// TIA Portal project "AB" (V15.1)

(* hardware
DEVICE "S71500/ET200MP station_1"  S7-1500 station
   slot 0: "导轨_0"  Rack  6ES7 590-1***0-0AA0
   slot 0: "PS 25W 24VDC_1"  PS 25W 24VDC  6ES7 505-0KA00-0AB0  V1.0
   slot 1: "PLC_1"  CPU 1515-2 PN  6ES7 515-2AM01-0AB0  V2.6
      slot 3: "CPU 显示_1"  6ES7591-1BA00-0AA0
DEVICE "HMI_1"  TP900 Comfort
   slot 0: "HMI_1"  TP900 Comfort  6AV2 124-0JC01-0AX0  15.1.0.0
   slot 1: "HMI_RT_1"  TP900 Comfort  6AV2 124-0JC01-0AX0  15.1.0.0
   slot 5: "HMI_1.IE_CP_1"  PROFINET Interface  15.0.1.0
      slot 1: "PROFINET Interface_1"  PROFINET Interface
         slot 1: "Port_1"  Port
         slot 2: "Port_2"  Port
   slot 7: "HMI_1.MPI/DP_CP_1"  MPI/DP Interface  15.0.1.0
*)

// ===== PLC "PLC_1"  CPU 1515-2 PN =====

VAR_GLOBAL   // PLC tag table "默认变量表"
   "System_Byte" AT %MB1 : Byte;
   "FirstScan" AT %M1.0 : Bool;
   "DiagStatusUpdate" AT %M1.1 : Bool;
   "AlwaysTRUE" AT %M1.2 : Bool;
   "AlwaysFALSE" AT %M1.3 : Bool;
   "Clock_Byte" AT %MB0 : Byte;
   "Clock_10Hz" AT %M0.0 : Bool;
   "Clock_5Hz" AT %M0.1 : Bool;
   "Clock_2.5Hz" AT %M0.2 : Bool;
   "Clock_2Hz" AT %M0.3 : Bool;
   "Clock_1.25Hz" AT %M0.4 : Bool;
   "Clock_1Hz" AT %M0.5 : Bool;
   "Clock_0.625Hz" AT %M0.6 : Bool;
   "Clock_0.5Hz" AT %M0.7 : Bool;
END_VAR

TYPE "Motor"
   STRUCT
      运行时间 : Time;   // 电机连续运行时间
      输出频率 : Real;   // 电机变频器当前输出频率
      A相电压 : Real;   // 变频器当前A相电压
      B相电压 : Real;   // 变频器当前B相电压
      C相电压 : Real;   // 变频器当前C相电压
      A相电流 : Real;   // 变频器当前A相电流
      B相电流 : Real;   // 变频器当前B相电流
      C相电流 : Real;   // 变频器当前C相电流
      启动 : Bool;   // 启动指令
      停止 : Bool;   // 停止指令
   END_STRUCT;
END_TYPE

DATA_BLOCK "_DeBug"   // DB1
{ S7_Optimized_Access := 'FALSE' }
VERSION : 0.1
   VAR
      IN : Word;
      max : Real;
      min : Real;
      amax : Int;
      amin : Int;
      error : Bool;
      status : Word;
      ret : Real;
      "1err" : Bool;
      "1sta" : Word;
      "1ot" : Word;
      计数 : Bool;
      temp : Array[0..1] of Bool;
      次数 : Int;
   END_VAR
BEGIN
END_DATA_BLOCK

// folder: 500 Communication

DATA_BLOCK "ConnectSet"   // DB501
{ S7_Optimized_Access := 'FALSE' }
VERSION : 0.1
   VAR
      connect : TCON_IP_v4;
   END_VAR
BEGIN
   connect.InterfaceId := 64;
   connect.ID := 1;
   connect.LocalPort := 502;
END_DATA_BLOCK

// folder: 500 Communication/PLCtoUpper

DATA_BLOCK "CommData_0x"   // DB503
{ S7_Optimized_Access := 'FALSE' }
VERSION : 0.1
   VAR
      "1-1#阀门" : Bool;   // 00001
      "1-2#阀门" : Bool;   // 00002
      "1-3#阀门" : Bool;   // 00003
      "1-4#阀门" : Bool;   // 00004
      "2-1#阀门" : Bool;   // 00005
      "2-2#阀门" : Bool;   // 00006
      "2-3#阀门" : Bool;   // 00007
      "2-4#阀门" : Bool;   // 00008
      "1#电机启动" : Bool;   // 00009
      "1#电机停止" : Bool;   // 00010
      "2#电机启动" : Bool;   // 00011
      "2#电机停止" : Bool;   // 00012
   END_VAR
BEGIN
END_DATA_BLOCK

DATA_BLOCK "CommData_4x"   // DB504
{ S7_Optimized_Access := 'FALSE' }
VERSION : 0.1
   VAR
      "1#电机" : Struct
         输出频率 : Real;   // 电机变频器当前输出频率
         A相电压 : Real;   // 变频器当前A相电压
         B相电压 : Real;   // 变频器当前B相电压
         C相电压 : Real;   // 变频器当前C相电压
         A相电流 : Real;   // 变频器当前A相电流
         B相电流 : Real;   // 变频器当前B相电流
         C相电流 : Real;   // 变频器当前C相电流
      END_STRUCT;
      "2#电机" : Struct
         输出频率 : Real;   // 电机变频器当前输出频率
         A相电压 : Real;   // 变频器当前A相电压
         B相电压 : Real;   // 变频器当前B相电压
         C相电压 : Real;   // 变频器当前C相电压
         A相电流 : Real;   // 变频器当前A相电流
         B相电流 : Real;   // 变频器当前B相电流
         C相电流 : Real;   // 变频器当前C相电流
      END_STRUCT;
      "1#电机运行时间" : Time;   // 40028
      "2#电机运行时间" : Time;   // 40030
   END_VAR
BEGIN
END_DATA_BLOCK

// folder: 500 Communication/PLCtoUpper/IDBs

DATA_BLOCK "块_1_IDB"   // DB2
{ S7_Optimized_Access := 'TRUE' }
VERSION : 0.1
// stored: InstanceOfName 块_1
"块_1"
BEGIN
END_DATA_BLOCK

// folder: (top level)

ORGANIZATION_BLOCK "Main"   // OB1, LAD, ProgramCycle
TITLE = "Main Program Sweep (Cycle)"
{ S7_Optimized_Access := 'TRUE' }
VERSION : 0.1
   VAR_INPUT
      Initial_Call : Bool;   // Initial call of this OB
      Remanence : Bool;   // =True, if remanent data are available
   END_VAR
   VAR_TEMP   // added for the SCL form of the ladder/FBD networks
      _w1 : Bool;
   END_VAR
BEGIN

REGION Network 1
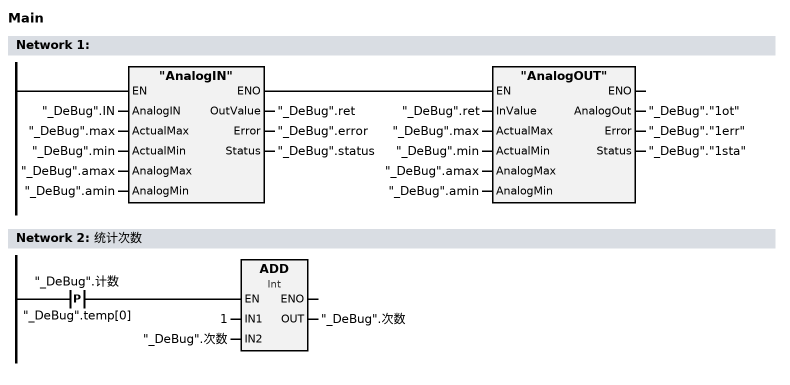
   RUNG wire#powerrail
      "AnalogIN"(AnalogIN := "_DeBug".IN, ActualMax := "_DeBug".max, ActualMin := "_DeBug".min, AnalogMax := "_DeBug".amax, AnalogMin := "_DeBug".amin, OutValue => "_DeBug".ret, Error => "_DeBug".error, Status => "_DeBug".status)
      "AnalogOUT"(InValue := "_DeBug".ret, ActualMax := "_DeBug".max, ActualMin := "_DeBug".min, AnalogMax := "_DeBug".amax, AnalogMin := "_DeBug".amin, AnalogOut => "_DeBug"."1ot", Error => "_DeBug"."1err", Status => "_DeBug"."1sta")
   END_RUNG
   // the same network as SCL:
   "AnalogIN"(AnalogIN := "_DeBug".IN,
              ActualMax := "_DeBug".max,
              ActualMin := "_DeBug".min,
              AnalogMax := "_DeBug".amax,
              AnalogMin := "_DeBug".amin,
              OutValue => "_DeBug".ret,
              Error => "_DeBug".error,
              Status => "_DeBug".status,
              ENO => #_w1);
   IF #_w1 THEN
       "AnalogOUT"(InValue := "_DeBug".ret,
                   ActualMax := "_DeBug".max,
                   ActualMin := "_DeBug".min,
                   AnalogMax := "_DeBug".amax,
                   AnalogMin := "_DeBug".amin,
                   AnalogOut => "_DeBug"."1ot",
                   Error => "_DeBug"."1err",
                   Status => "_DeBug"."1sta");
   END_IF;
END_REGION

REGION Network 2: 统计次数
   RUNG wire#powerrail
      P_Contact(operand := "_DeBug".计数, bit := "_DeBug".temp[0])
      { S7_Templates := "SrcType := Int" } Add(in1 := 1, in2 := "_DeBug".次数, out => "_DeBug".次数)
   END_RUNG
   // the same network as SCL:
   #_w1 := "_DeBug".计数 AND NOT "_DeBug".temp[0];   // rising edge of "_DeBug".计数
   "_DeBug".temp[0] := "_DeBug".计数;
   IF #_w1 THEN "_DeBug".次数 := 1 + "_DeBug".次数; END_IF;
END_REGION
END_ORGANIZATION_BLOCK

// folder: 000 Initialization

ORGANIZATION_BLOCK "Startup"   // OB100, LAD, Startup
TITLE = "Complete Restart"
{ S7_Optimized_Access := 'TRUE' }
VERSION : 0.1
   VAR_INPUT
      LostRetentive : Bool;   // True if retentive data are lost
      LostRTC : Bool;   // True if date and time are lost
   END_VAR
BEGIN
END_ORGANIZATION_BLOCK

// folder: 500 Communication

ORGANIZATION_BLOCK "Comm"   // OB123, LAD, ProgramCycle
TITLE = "Main Program Sweep (Cycle)"
{ S7_Optimized_Access := 'TRUE' }
VERSION : 0.1
   VAR_INPUT
      Initial_Call : Bool;   // Initial call of this OB
      Remanence : Bool;   // =True, if remanent data are available
   END_VAR
BEGIN

REGION Network 1
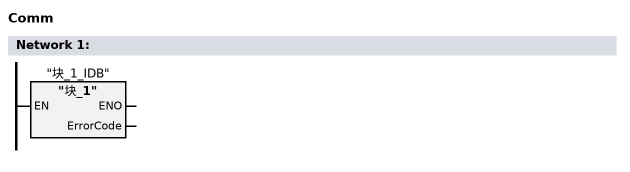
   RUNG wire#powerrail
      "块_1_IDB"(ErrorCode =>)
   END_RUNG
   // the same network as SCL:
   "块_1_IDB"();   // "块_1"
END_REGION
END_ORGANIZATION_BLOCK

// folder: 500 Communication/PLCtoUpper

FUNCTION_BLOCK "块_1"   // FB501, LAD
{ S7_Optimized_Access := 'TRUE' }
VERSION : 0.1
   VAR_OUTPUT
      ErrorCode : Word;
   END_VAR
   VAR
      MB_SERVER_Instance : MB_SERVER;
      pulses : Array[0..9] of Bool;
   END_VAR
   VAR_TEMP   // added for the SCL form of the ladder/FBD networks
      _w1 : Bool;
   END_VAR
BEGIN

REGION Network 1
   // 1、当在mod_server背景数据块里用data_area_array参数规定缓存区域后，MB_HOLD_REG参数就无效，随便填写一个没用使用的区域
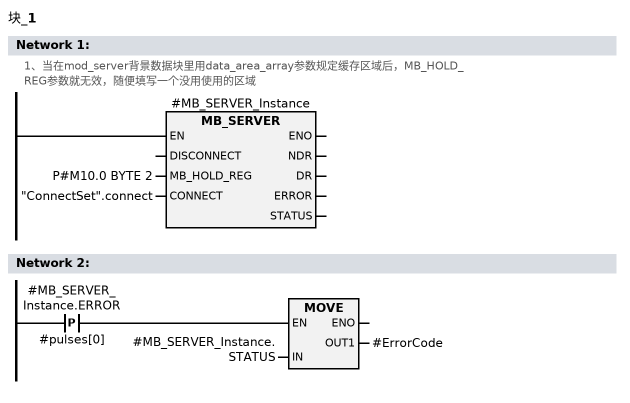
   #MB_SERVER_Instance(MB_HOLD_REG := P#M10.0 BYTE 2, CONNECT := "ConnectSet".connect);   // MB_SERVER
END_REGION

REGION Network 2
   RUNG wire#powerrail
      P_Contact(operand := #MB_SERVER_Instance.ERROR, bit := #pulses[0])
      Move(in := #MB_SERVER_Instance.STATUS, out1 => #ErrorCode)
   END_RUNG
   // the same network as SCL:
   #_w1 := #MB_SERVER_Instance.ERROR AND NOT #pulses[0];   // rising edge of #MB_SERVER_Instance.ERROR
   #pulses[0] := #MB_SERVER_Instance.ERROR;
   IF #_w1 THEN #ErrorCode := #MB_SERVER_Instance.STATUS; END_IF;
END_REGION
END_FUNCTION_BLOCK

// folder: 999 Basic/AnalogFunc

FUNCTION_BLOCK "AnalogAlarm"   // FB1003, LAD
{ S7_Optimized_Access := 'TRUE' }
VERSION : 0.1
   VAR_INPUT
      输入值 : Real;
      低低限值 : Real;
      低限值 : Real;
      高限值 : Real;
      高高限值 : Real;
      报警延迟时间 : Time := T#2s;
   END_VAR
   VAR_OUTPUT
      低低报警 : Bool;
      低报警 : Bool;
      高报警 : Bool;
      高高报警 : Bool;
      Error : Bool;
      Status : Bool;
   END_VAR
BEGIN
END_FUNCTION_BLOCK

FUNCTION "AnalogIN" : Void   // FC1001, SCL
{ S7_Optimized_Access := 'TRUE' }
VERSION : 0.1
   VAR_INPUT
      AnalogIN : Word;   // 模拟量值接口输入
      ActualMax : Real;   // 实际工程值最大值
      ActualMin : Real;   // 实际工程值最小值
      AnalogMax : Int;   // 模拟量数字值最大值
      AnalogMin : Int;   // 模拟量数字值最小值
   END_VAR
   VAR_OUTPUT
      OutValue : Real;   // 转换后的输出工程值
      Error : Bool;   // 是否错误
      Status : Word;   // 状态字
   END_VAR
   VAR_TEMP
      IntAnalog : Int;   // 暂时保存的整数类型输入值
   END_VAR
   VAR CONSTANT
      NOERROR : Word := 16#0000;   // 命令完成，没有警告，也没有进一步的详细信息
      BUSY : Word := 16#7002;   // 在命令激活后续调用中执行期间，无详细信息提供
      ACTUALVALUEERROR : Word := 16#8201;   // 参数设定错误（实际工程值设定最小值大于最大值）
      ANALOGVALUEERROR : Word := 16#8301;   // 参数设定错误（模拟量数字值设定最小值大于最大值）
   END_VAR
BEGIN
   REGION 初始化输出值
     #Error := FALSE;
     #Status := #NOERROR;
   END_REGION
   REGION 检测输入值是否正确，若不正确则直接退出

     IF #ActualMax < #ActualMin THEN
       #Error := True;
       #Status := #ACTUALVALUEERROR;
       RETURN;
     END_IF;
     IF #AnalogMax < #AnalogMin THEN
       #Error := True;
       #Status := #ANALOGVALUEERROR;
       RETURN;
     END_IF;
   END_REGION
   REGION 转换值
     #Status := #BUSY;
     #IntAnalog:= WORD_TO_INT(#AnalogIN);
     #OutValue:= SCALE_X(MIN:=#ActualMin, VALUE:=NORM_X(MIN := #AnalogMin, VALUE := #IntAnalog, MAX := #AnalogMax), MAX:=#ActualMax);
   END_REGION
END_FUNCTION

FUNCTION "AnalogOUT" : Void   // FC1002, SCL
{ S7_Optimized_Access := 'TRUE' }
VERSION : 0.1
   VAR_INPUT
      InValue : Real;   // 工程值输入
      ActualMax : Real;   // 实际工程值最大值
      ActualMin : Real;   // 实际工程值最小值
      AnalogMax : Int;   // 模拟量数字值最大值
      AnalogMin : Int;   // 模拟量数字值最小值
   END_VAR
   VAR_OUTPUT
      AnalogOut : Word;   // 模拟数字值输出
      Error : Bool;   // 错误位
      Status : Word;   // 状态字
   END_VAR
   VAR CONSTANT
      NOERROR : Word := 16#0000;   // 命令完成，没有警告，也没有进一步的详细信息
      BUSY : Word := 16#7002;   // 在命令激活后续调用中执行期间，无详细信息提供
      ACTUALVALUEERROR : Word := 16#8201;   // 参数设定错误（实际工程值设定最小值大于最大值）
      ANALOGVALUEERROR : Word := 16#8301;   // 参数设定错误（模拟量数字值设定最小值大于最大值）
   END_VAR
BEGIN
   REGION 初始化输出值
     #Error := FALSE;
     #Status := #NOERROR;
   END_REGION
   REGION 检测输入值是否正确，若不正确则直接退出

     IF #ActualMax < #ActualMin THEN
       #Error := True;
       #Status := #ACTUALVALUEERROR;
       RETURN;
     END_IF;
     IF #AnalogMax < #AnalogMin THEN
       #Error := True;
       #Status := #ANALOGVALUEERROR;
       RETURN;
     END_IF;
   END_REGION
   REGION 转换值
     #Status := #BUSY;
     #AnalogOut:= INT_TO_WORD(SCALE_X(MIN := #AnalogMin, VALUE := NORM_X(MIN := #ActualMin, VALUE := #InValue, MAX := #ActualMax), MAX := #AnalogMax));
   END_REGION
END_FUNCTION

(* ===== HMI "HMI_RT_1" =====
system functions are stored by id; their names below are inferred from use
connection "HMI_连接_1": ETHERNET, S7_1500_OMS

HMI tags "默认变量表"
   "Tag_ScreenNumber" : UInt, internal
   "CommData_0x_1-1#阀门" : Bool = PLC CommData_0x.1-1#阀门 AT %DB503.DBX0.0, 1 s
   "_DeBug_IN" : Word = PLC _DeBug.IN AT %DB1.DBW0, 1 s
   "_DeBug_amax" : Int = PLC _DeBug.amax AT %DB1.DBW10, 1 s

discrete alarms
   1: '', class Errors, trigger "_DeBug_IN" bit 0

analog alarms
   1: '', class Errors, trigger "_DeBug_amax"

screen "根画面" 800x420, template "模板_1"
   on GenerateScreen: SetTag("Tag_ScreenNumber", 1)
   AlarmView "报警视图_1" at 0,0 size 794x351

Template "模板_1" 800x420
   Button "退出" at 720,360 size 78x58; TextOff '退出'; PictureOff "ExitRuntime_TP900_Comfort_TR"; PictureOn "ExitRuntime_TP900_Comfort_TR"
      on Release: StopRuntime(0)
   Button "Template_Button" at 640,360 size 78x58; TextOff 'Text'
   Button "Template_Button_1" at 560,360 size 78x58; TextOff 'Text'
   Button "Template_Button_2" at 480,360 size 78x58; TextOff 'Text'
   Button "Template_Button_3" at 400,360 size 78x58; TextOff 'Text'
   Button "Template_Button_4" at 321,360 size 78x58; TextOff 'Text'
   Button "Template_Button_5" at 241,360 size 78x58; TextOff 'Text'
   Button "Template_Button_6" at 161,360 size 78x58; TextOff 'Text'
   Button "报警" at 81,360 size 78x58; TextOff '报警'; PictureOff "AlarmDisplay_TP900_Comfort_TR"; PictureOn "AlarmDisplay_TP900_Comfort_TR"
      on Release: function_ef3f5d25("报警窗口_Unacknowledged", -1)
   Button "起始画面" at 1,360 size 78x58; TextOff '起始画面'; PictureOff "NavigateHome_TP900_Comfort_TR"; PictureOn "NavigateHome_TP900_Comfort_TR"
      on Release: ActivateScreen("根画面", 0)
*)